(* LS Electric XG5000 project: XMC_SingleAxis_FBs *)
(* sample programs for single axis function blocks. *)
(* PLC LSPLC *)
(* module base 0 slot 0: Input/Output Module:XMC-DN24 (DC 24V Input 8Points/TR output 16Points) *)
(* module base 0 slot 1: Internal Analog Input/Output:XMF-AH04E (A/D voltage/current 2 channels, D/A voltage 2 channels) *)
(* task Periodic Task: Kind=2 *)
(* task Initialization Task: Kind=1 *)
(* task NC Program: Kind=6 *)
VAR_GLOBAL
    ContinuousRelative_INST : MC_MOVECONTINUOUSRELATIVE; (* MC_MoveContinuousRelative fb *)
    Relative_INST : MC_MOVECONTINUOUSRELATIVE; (* MC_MoveContinuousRelative fb *)
END_VAR

PROGRAM ECAT_Connect_Example (* task: Scan Program *)
(* example of LS_Connect and LS_Disconnect function blocks *)
VAR
    Execute_Connect : BOOL; (* Execute LS_Connect function block *)
    Execute_Disconnect : BOOL; (* Execute LS_Disconnect *)
    INST_LS_CONNECT : LS_CONNECT; (* Instance of LS_Connect function block *)
    INST_LS_DISCONNECT : LS_DISCONNECT; (* LS_Disconnect function block instance *)
END_VAR
(* AutomationDirect.com has provided this code for convenience. This sample code is provided "as-is" with no expressed or implied warranty. 
 If the end user includes any of the sample code (in whole or part), it is the user's responsibility to completely modify, integrate, and test any code to ensure it meets all system and 
 safety requirements for the intended application or system. *)

//Example of LS_Connect Function block to connect EtherCAT network
INST_LS_CONNECT(Execute:=Execute_Connect, ErrorID=>INST_LS_CONNECT.ErrorID);

//Example of LS_Disconnect Function block to disconnect the EtherCAT network
INST_LS_DISCONNECT(Execute:=Execute_Disconnect, ErrorID=>INST_LS_DISCONNECT.ErrorID);
END_PROGRAM

PROGRAM MC_Power_Example (* task: Scan Program *)
(* ST example of MC_Power *)
VAR
    Axis1 : UINT; (* axis 1 reference variable *)
    Enable_Power : BOOL; (* command to enable axis power *)
    INST_MC_POWER : MC_POWER; (* MC_Power fb *)
END_VAR
//Set Axis 1 reference
Axis1 := 1;

//Example MC_Power FB.  Check that axis is ready
IF (_AX01_RDY) THEN
	INST_MC_POWER(Enable:=Enable_Power, Axis:=Axis1, ErrorID=>INST_MC_POWER.ErrorID);
END_IF;
END_PROGRAM

PROGRAM Home_Example (* task: Scan Program *)
(* ST example of MC_Home and LS_Home *)
VAR
    Axis1 : UINT; (* axis1 reference variable *)
    Execute_LSHome : BOOL; (* execute LS_Home fb *)
    Execute_MCHome : BOOL; (* execute MC_Home fb *)
    INST_LS_HOME : LS_HOME; (* LS_Home function block *)
    INST_MC_HOME : MC_HOME; (* MC_Home fb *)
END_VAR
//Set Axis1 reference variable
Axis1 := 1;

//check that axis 1 is ready
IF (_AX01_RDY) AND (_AX01_SV_ON) THEN
	
	//Example MC_Home fb
	INST_MC_HOME(Execute:=Execute_MCHome, Axis:=Axis1, Position:=INST_MC_HOME.Position, BufferMode:=0, ErrorID=>INST_MC_HOME.ErrorID);
	
	//Example LS_Home fb
	INST_LS_HOME(Execute:=Execute_LSHome, Axis:=Axis1, Position:=INST_LS_HOME.Position, HomingMethod:=INST_LS_HOME.HomingMethod, 
		SwitchSearchSpeed:=INST_LS_HOME.SwitchSearchSpeed, ZeroSearchSpeed:=INST_LS_HOME.ZeroSearchSpeed, HomingAcc:=INST_LS_HOME.HomingAcc, 
		HomeOffset:=INST_LS_HOME.HomeOffset, DoneBehavior:=INST_LS_HOME.DoneBehavior, BufferMode:=0, ErrorID=>INST_LS_HOME.ErrorID);
END_IF;
END_PROGRAM

PROGRAM MCStop_MCHalt_Example (* task: Scan Program *)
(* ST example for MC_Stop and MC_Halt fb *)
VAR
    Axis1 : UINT; (* reference variable for axis1 *)
    Execute_MCHalt : BOOL; (* Execute MC_Halt fb *)
    Execute_MCStop : BOOL; (* execute MC_Stop fb *)
    INST_MC_HALT : MC_HALT; (* MC_Halt fb *)
    INST_MC_STOP : MC_STOP; (* MC_Stop function block *)
END_VAR
//Set reference for axis
Axis1 := 1;

//check that axes are ready
IF (_AX01_RDY) AND (_AX01_SV_ON) THEN
	//Example of MC_Stop fb
	INST_MC_STOP(Execute:=Execute_MCStop, Axis:=Axis1, Deceleration:=50000.0, Jerk:=1000.0, ErrorID=>INST_MC_STOP.ErrorID);
	
	//Example of MC_Halt fb
	INST_MC_HALT(Execute:=Execute_MCHalt, Axis:=Axis1, Deceleration:=50000.0, Jerk:=1000.0, BufferMode:=0,ErrorID=>INST_MC_HALT.ErrorID);
END_IF;
END_PROGRAM

PROGRAM Read_Status_FBs (* task: Scan Program *)
(* ST example for MC fbs that read axis status *)
VAR
    Axis1 : UINT; (* reference for axis 1 *)
    Enable_ReadActualPosition : BOOL; (* enable MC_ReadActualPosition fb *)
    Enable_ReadActualTorque : BOOL; (* Enable MC_ReadActualTorque fb *)
    Enable_ReadActualVelocity : BOOL; (* enable MC_ReadActualVelocity fb *)
    Enable_ReadCommandedPosition : BOOL; (* enable MC_ReadCommandedPosition *)
    Enable_ReadCommandedTorque : BOOL; (* enable MC_ReadCommandedTorque fb *)
    Enable_ReadCommandedVelocity : BOOL; (* enable MC_ReadCommandedVelocity fb *)
    Enable_ReadMotionInfo : BOOL; (* Enable MC_ReadMotionInfo fb *)
    INST_READACTUALPOSITION : MC_READACTUALPOSITION; (* MC_ReadActualPosition fb *)
    INST_READACTUALTORQUE : MC_READACTUALTORQUE; (* MC_ReadActualTorque function block *)
    INST_READACTUALVELOCITY : MC_READACTUALVELOCITY; (* MC_ReadActualVelocity fb *)
    INST_READCOMMANDEDPOSITION : MC_READCOMMANDEDPOSITION; (* MC_ReadCommandedPosition fb *)
    INST_READCOMMANDEDTORQUE : MC_READCOMMANDEDTORQUE; (* MC_ReadCommandedTorque fb *)
    INST_READCOMMANDEDVELOCITY : MC_READCOMMANDEDVELOCITY; (* MC_ReadCommandedVelocity fb *)
    INST_READMOTIONINFO : MC_READMOTIONINFO; (* MC_ReadMotionInfo fb *)
END_VAR
//Set Axis Reference
Axis1 := 1;

IF (_AX01_RDY) THEN
	//Example of MC_ReadMotionInfo
	INST_READMOTIONINFO(Enable:=Enable_ReadMotionInfo, Axis:=Axis1, ParameterNumber:=INST_READMOTIONINFO.ParameterNumber, ErrorID=>INST_READMOTIONINFO.ErrorID);
	
	//Example of MC_ReadActualPosition
	INST_READACTUALPOSITION(Enable:=Enable_ReadActualPosition, Axis:=Axis1, ErrorID=>INST_READACTUALPOSITION.ErrorID);
	
	//Example of MC_ReadActualVelocity
	INST_READACTUALVELOCITY(Enable:=Enable_ReadActualVelocity, Axis:=Axis1, ErrorID=>INST_READACTUALVELOCITY.ErrorID);
	
	//Example of MC_ReadActualTorque
	INST_READACTUALTORQUE(Enable:=Enable_ReadActualTorque, Axis:=Axis1, ErrorID=>INST_READACTUALTORQUE.ErrorID);
	
	//Example of MC_ReadCommandedPosition
	INST_READCOMMANDEDPOSITION(Enable:=Enable_ReadCommandedPosition, Axis:=Axis1,ErrorID=>INST_READCOMMANDEDPOSITION.ErrorID);
	
	//Example of MC_ReadCommandedVelocity
	INST_READCOMMANDEDVELOCITY(Enable:=Enable_ReadCommandedVelocity, Axis:=Axis1, ErrorID=>INST_READCOMMANDEDVELOCITY.ErrorID);
	
	//Example MC_ReadCommandedTorque
	INST_READCOMMANDEDTORQUE(Enable:=Enable_ReadCommandedTorque, Axis:=Axis1, ErrorID=>INST_READCOMMANDEDTORQUE.ErrorID);
	
END_IF;
END_PROGRAM

PROGRAM MC_Reset_Example (* task: Scan Program *)
(* ST example for MC_Reset & MC_Reset2 *)
VAR
    Axis1 : UINT; (* reference variable for axis1 *)
    Execute_MCReset : BOOL; (* execute MC_Reset fb *)
    Execute_MCReset2 : BOOL; (* Execute MC_Reset2 fb *)
    INST_MC_RESET : MC_RESET; (* MC_Reset fb *)
    INST_MC_RESET2 : MC_RESET2; (* MC_Reset2 fb *)
END_VAR
//Set Axis Reference
Axis1 := 1;

IF (_AX01_RDY) THEN
	//Example of MC_Reset
	INST_MC_RESET(Execute:=Execute_MCReset, Axis:=Axis1, ErrorType:=INST_MC_RESET.ErrorType, ErrorID=>INST_MC_RESET.ErrorID);
	
	INST_MC_RESET2(Execute:=Execute_MCReset2, Axis:=Axis1, ErrorType:=INST_MC_RESET2.ErrorType, ErrorID=>INST_MC_RESET2.ErrorID);
	
END_IF;
END_PROGRAM

PROGRAM MC_MoveAbsolute_Example (* task: Scan Program *)
(* example of MC_MoveAbsolute *)
VAR
    Axis1 : UINT; (* axis 1 reference variable *)
    Execute_MoveAbsolute : BOOL; (* execute MC_MoveAbsolute *)
    INST_MOVEABSOLUTE : MC_MOVEABSOLUTE; (* MC_MoveAbsolute fb *)
END_VAR
//Set axis reference
Axis1 := 1;

IF (_AX01_RDY) AND (_AX01_SV_ON) AND (_AX01_HOME_CMPL) THEN
	//Example of MC_MoveAbsolute
	INST_MOVEABSOLUTE(Execute:=Execute_MoveAbsolute, Axis:=Axis1, ContinuousUpdate:=0, Position:=INST_MOVEABSOLUTE.Position, 
		Velocity:=INST_MOVEABSOLUTE.Velocity, Acceleration:=INST_MOVEABSOLUTE.Acceleration, Deceleration:=INST_MOVEABSOLUTE.Deceleration, 
		Jerk:=INST_MOVEABSOLUTE.Jerk, Direction:=INST_MOVEABSOLUTE.Direction, BufferMode:=0, ErrorID=>INST_MOVEABSOLUTE.ErrorID);
END_IF;
END_PROGRAM

PROGRAM MC_MoveRelative_Example (* task: Scan Program *)
(* ST example for MC_MoveRelative fb *)
VAR
    Axis1 : UINT; (* reference for Axis1 *)
    Execute_MoveRelative : BOOL; (* execute MC_MoveRelative fb *)
    INST_MOVERELATIVE : MC_MOVERELATIVE; (* MC_MoveRelative fb *)
END_VAR
//Set axis reference
Axis1 := 1;

IF (_AX01_RDY) AND (_AX01_SV_ON) THEN
	//Example of MC_MoveRelative
	INST_MOVERELATIVE(Execute:=Execute_MoveRelative, Axis:=Axis1, ContinuousUpdate:=0, Distance:=INST_MOVERELATIVE.Distance,
		 Velocity:=INST_MOVERELATIVE.Velocity, Acceleration:=INST_MOVERELATIVE.Acceleration, Deceleration:=INST_MOVERELATIVE.Deceleration, 
		 Jerk:=INST_MOVERELATIVE.Jerk, BufferMode:=0, ErrorID=>INST_MOVERELATIVE.ErrorID);	
END_IF;
END_PROGRAM

PROGRAM MC_MoveAdditive_Example (* task: Scan Program *)
(* ST example for MC_MoveAdditive fb *)
VAR
    Axis1 : UINT; (* axis 1 reference variable *)
    Execute_MoveAdditive : BOOL; (* execute MC_MoveAdditive fb *)
    INST_MOVEADDITIVE : MC_MOVEADDITIVE; (* MC_MoveAdditive fb *)
END_VAR
//Set axis reference
Axis1 := 1;

IF (_AX01_RDY) AND (_AX01_SV_ON) AND (_AX01_HOME_CMPL) THEN
	//Example of MC_MoveAdditive
	INST_MOVEADDITIVE(Execute:=Execute_MoveAdditive, Axis:=Axis1, ContinuousUpdate:=0, Distance:=INST_MOVEADDITIVE.Distance, 
		Velocity:=INST_MOVEADDITIVE.Velocity, Acceleration:=INST_MOVEADDITIVE.Acceleration, Deceleration:=INST_MOVEADDITIVE.Deceleration, 
		Jerk:=INST_MOVEADDITIVE.Jerk, BufferMode:=0, ErrorID=>INST_MOVEADDITIVE.ErrorID);
END_IF;
END_PROGRAM

PROGRAM MC_MoveVelocity_Example (* task: Scan Program *)
(* ST example for MC_MoveVelocity fb *)
VAR
    Axis1 : UINT; (* axis 1 reference variable *)
    Execute_MoveVelocity : BOOL; (* execute MC_MoveVelocity fb *)
    INST_MOVEVELOCITY : MC_MOVEVELOCITY; (* MC_MoveVelocity fb *)
END_VAR
//Set axis reference
Axis1 := 1;

IF (_AX01_RDY) AND (_AX01_SV_ON)  THEN
	//Example MC_MoveVelocity fb
	INST_MOVEVELOCITY(Execute:=Execute_MoveVelocity, Axis:=Axis1, ContinuousUpdate:=0, Velocity:=INST_MOVEVELOCITY.Velocity, 
		Acceleration:=INST_MOVEVELOCITY.Acceleration, Deceleration:=INST_MOVEVELOCITY.Deceleration, Jerk:=INST_MOVEVELOCITY.Jerk, 
		Direction:=INST_MOVEVELOCITY.Direction, BufferMode:=0, ErrorID=>INST_MOVEVELOCITY.ErrorID);
END_IF;
END_PROGRAM

PROGRAM MC_MoveContinuousAbsolute_Example (* task: Scan Program *)
(* ST example of MC_MoveContinuousAbsolute fb *)
VAR
    Axis1 : UINT; (* axis 1 reference variable *)
    Execute_MoveContAbs : BOOL; (* execute MC_MoveContinuousAbsolute fb *)
    INST_MOVECONTINUOUSABSOLUTE : MC_MOVECONTINUOUSABSOLUTE; (* MC_MoveContinuousAbsolute fb *)
END_VAR
//Set axis reference
Axis1 := 1;

IF (_AX01_RDY) AND (_AX01_SV_ON)  AND (_AX01_HOME_CMPL) THEN
	//Example MC_MoveContinuousAbsolute fb
	INST_MOVECONTINUOUSABSOLUTE(Execute:=Execute_MoveContAbs, Axis:=Axis1, ContinuousUpdate:=0, Position:=INST_MOVECONTINUOUSABSOLUTE.Position, 
		EndVelocity:=INST_MOVECONTINUOUSABSOLUTE.EndVelocity, Velocity:=INST_MOVECONTINUOUSABSOLUTE.Velocity, Acceleration:=INST_MOVECONTINUOUSABSOLUTE.Acceleration, 
		Deceleration:=INST_MOVECONTINUOUSABSOLUTE.Deceleration, Jerk:=INST_MOVECONTINUOUSABSOLUTE.Jerk, Direction:=INST_MOVECONTINUOUSABSOLUTE.Direction, 
		BufferMode:=0, ErrorID=>INST_MOVECONTINUOUSABSOLUTE.ErrorID);
END_IF;
END_PROGRAM

PROGRAM MC_MoveContinuousRelative_Example (* task: Scan Program *)
(* ST example for MC_MoveContinuousRelative fb *)
VAR
    Axis1 : UINT; (* axis 1 reference variable *)
    Execute_MoveContRel : BOOL; (* execute MC_MoveContinuousRelative fb *)
    INST_MOVECONTINUOUSRELATIVE : MC_MOVECONTINUOUSRELATIVE; (* MC_MoveContinuousRelative fb *)
END_VAR
//Set axis reference
Axis1 := 1;

IF (_AX01_RDY) AND (_AX01_SV_ON) THEN
	//Example MC_MoveContinuousRelative fb
	INST_MOVECONTINUOUSRELATIVE(Execute:=Execute_MoveContRel, Axis:=Axis1, ContinuousUpdate:=0, Distance:=INST_MOVECONTINUOUSRELATIVE.Distance, 
		EndVelocity:=INST_MOVECONTINUOUSRELATIVE.EndVelocity, Velocity:=INST_MOVECONTINUOUSRELATIVE.Velocity, Acceleration:=INST_MOVECONTINUOUSRELATIVE.Acceleration, 
		Deceleration:=INST_MOVECONTINUOUSRELATIVE.Deceleration, Jerk:=INST_MOVECONTINUOUSRELATIVE.Jerk, 
		BufferMode:=0, ErrorID=>INST_MOVECONTINUOUSRELATIVE.ErrorID);
END_IF;
END_PROGRAM

PROGRAM MC_TorqueControl_Example (* task: Scan Program *)
(* ST example for MC_TorqueControl fb *)
VAR
    Axis1 : UINT; (* axis 1 reference variable *)
    Execute_TrqControl : BOOL; (* Execute MC_TorqueControl fb *)
    INST_TORQUECONTROL : MC_TORQUECONTROL; (* MC_TorqueControl fb *)
END_VAR
//Set axis reference
Axis1 := 1;

IF (_AX01_RDY) AND (_AX01_SV_ON) THEN
	//Example MC_TorqueControl fb
	INST_TORQUECONTROL(Execute:=Execute_TrqControl, Axis:=Axis1, ContinuousUpdate:=0, Torque:=INST_TORQUECONTROL.Torque, 
		TorqueRamp:=INST_TORQUECONTROL.TorqueRamp, Velocity:=INST_TORQUECONTROL.Velocity, Acceleration:=INST_TORQUECONTROL.Acceleration, 
		Deceleration:=INST_TORQUECONTROL.Deceleration, Jerk:=INST_TORQUECONTROL.Jerk, Direction:=INST_TORQUECONTROL.Direction, 
		BufferMode:=0, ErrorID=>INST_TORQUECONTROL.ErrorID);
END_IF;
END_PROGRAM

PROGRAM MC_SetPosition_Example (* task: Scan Program *)
(* ST example of MC_SetPosition *)
VAR
    Axis1 : UINT; (* axis 1 reference variable *)
    Execute_SetPosition : BOOL; (* execute MC_SetPosition fb *)
    INST_SETPOSITION : MC_SETPOSITION; (* MC_SetPositionFB *)
END_VAR
//Set axis reference
Axis1 := 1;

IF (_AX01_RDY) AND (_AX01_SV_ON) THEN
	//Example MC_SetPosition fb
	INST_SETPOSITION(Execute:=Execute_SetPosition, Axis:=Axis1, Position:=INST_SETPOSITION.Position, Relative:=INST_SETPOSITION.Relative, 
		ExecutionMode:=INST_SETPOSITION.ExecutionMode, ErrorID=>INST_SETPOSITION.ErrorID);
END_IF;
END_PROGRAM

PROGRAM MC_SetOverride_Example (* task: Scan Program *)
(* ST example of MC_SetOverride fb *)
VAR
    Axis1 : UINT; (* axis 1 reference variable *)
    Execute_Override : BOOL; (* execute MC_SetOverride *)
    INST_SETOVERRIDE : MC_SETOVERRIDE; (* MC_SetOverride fb *)
END_VAR
//Set axis reference
Axis1 := 1;

IF (_AX01_RDY) AND (_AX01_SV_ON) THEN
	//Example MC_SetOverride fb
	INST_SETOVERRIDE(Enable:=Execute_Override, Axis:=Axis1, VelFactor:=INST_SETOVERRIDE.VelFactor, AccFactor:=INST_SETOVERRIDE.AccFactor, 
		JerkFactor:=INST_SETOVERRIDE.JerkFactor, ErrorID=>INST_SETOVERRIDE.ErrorID);
END_IF;
END_PROGRAM

PROGRAM Read_Write_Parameters (* task: Scan Program *)
(* ST example for MC_ReadParameter and MC_WriteParameter *)
VAR
    Axis1 : UINT; (* axis 1 reference variable *)
    Execute_Read : BOOL; (* Execute MC_ReadParameter fb *)
    Execute_Write : BOOL; (* execute MC_WriteParameter *)
    INST_READPARAMETER : MC_READPARAMETER; (* MC_ReadParameter fb *)
    INST_WRITEPARAMETER : MC_WRITEPARAMETER; (* MC_WriteParameter fb *)
END_VAR
//Set axis reference
Axis1 := 1;

IF (_AX01_RDY) THEN
	//Example of MC_ReadParameter fb
	INST_READPARAMETER(Enable:=Execute_Read, Axis:=Axis1, ParameterNumber:=INST_READPARAMETER.ParameterNumber, 
		ErrorID=>INST_READPARAMETER.ErrorID, Value=>INST_READPARAMETER.Value);
		
	
	//Example of MC_WriteParameter fb
	INST_WRITEPARAMETER(Execute:=Execute_Write, Axis:=Axis1, ParameterNumber:=INST_WRITEPARAMETER.ParameterNumber, Value:=INST_WRITEPARAMETER.Value, 
		ExecutionMode:=INST_WRITEPARAMETER.ExecutionMode, ErrorID=>INST_WRITEPARAMETER.ErrorID);	
		
END_IF;
END_PROGRAM

PROGRAM MC_TouchProbe_Example (* task: Scan Program *)
(* ST example of MC_TouchProbe and MC_TouchProbeEx *)
VAR
    Axis1 : UINT; (* axis 1 reference *)
    Execute_TouchProbe : BOOL; (* execute MC_TouchProbe *)
    Execute_TouchProveEx : BOOL; (* execute MC_TouchProbeEX fb *)
    INST_TOUCHPROBE : MC_TOUCHPROBE; (* MC_TouchProbe fb *)
    INST_TOUCHPROBEEX : MC_TOUCHPROBEEX; (* MC_TouchProbeEx fb *)
END_VAR
//Set axis reference
Axis1 := 1;

IF (_AX01_RDY) AND (_AX01_SV_ON) THEN
	//Example MC_TouchProbel fb
	INST_TOUCHPROBE(Execute:=Execute_TouchProbe, Axis:=Axis1, TriggerInput:=INST_TOUCHPROBE.TriggerInput, WindowOnly:=INST_TOUCHPROBE.WindowOnly, 
		FirstPosition:=INST_TOUCHPROBE.FirstPosition, LastPosition:=INST_TOUCHPROBE.LastPosition, 
		ErrorID=>INST_TOUCHPROBE.ErrorID, RecordedPosition=>INST_TOUCHPROBE.RecordedPosition);
		
	
	//Exampe of MC_TouchProbeEX fb
	INST_TOUCHPROBEEX(Execute:=Execute_TouchProveEx, Axis:=Axis1, TriggerInput:=INST_TOUCHPROBEEX.TriggerInput, TriggerMode:=INST_TOUCHPROBEEX.TriggerMode, 
		WindowOnly:=INST_TOUCHPROBEEX.WindowOnly, FirstPosition:=INST_TOUCHPROBEEX.FirstPosition, LastPosition:=INST_TOUCHPROBEEX.LastPosition, 
		ErrorID=>INST_TOUCHPROBEEX.ErrorID, RecordedPosition=>INST_TOUCHPROBEEX.RecordedPosition);
		
END_IF;
END_PROGRAM

PROGRAM MC_AbortTrigger_Example (* task: Scan Program *)
(* ST example MC_AbortTrigger fb *)
VAR
    Axis1 : UINT; (* axis 1 reference *)
    Execute_AbortTrigger : BOOL; (* execute MC_AbortTrigger fb *)
    INST_ABORTTRIGGER : MC_ABORTTRIGGER; (* MC_AbortTrigger fb *)
END_VAR
//Set axis reference
Axis1 := 1;

IF (_AX01_RDY) AND (_AX01_SV_ON) THEN
	//Example MC_AbortTrigger fb
	INST_ABORTTRIGGER(Execute:=Execute_AbortTrigger, Axis:=Axis1, TriggerInput:=INST_ABORTTRIGGER.TriggerInput, ErrorID=>INST_ABORTTRIGGER.ErrorID);
END_IF;
END_PROGRAM

PROGRAM MC_SuperImposed_Example (* task: Scan Program *)
(* ST example of MC_SuperImposed and MC_HaltSuperImposed *)
VAR
    Axis1 : UINT; (* axis 1 reference *)
    Execute_HaltSuperImposed : BOOL; (* execute MC_HaltSuperImposed fb *)
    Execute_SuperImposed : BOOL; (* execute MC_MoveSuperImposed *)
    INST_HALTSUPERIMPOSED : MC_HALTSUPERIMPOSED; (* MC_HaltSuperImposed *)
    INST_MOVESUPERIMPOSED : MC_MOVESUPERIMPOSED; (* MC_MoveSuperImposed fb *)
END_VAR
//Set axis reference
Axis1 := 1;

IF (_AX01_RDY) AND (_AX01_SV_ON) THEN
	//Example MC_MoveSuperImposed fb
	INST_MOVESUPERIMPOSED(Execute:=Execute_SuperImposed, Axis:=Axis1, ContinuousUpdate:=0, Distance:=INST_MOVESUPERIMPOSED.Distance, 
		VelocityDiff:=INST_MOVESUPERIMPOSED.VelocityDiff, Acceleration:=INST_MOVESUPERIMPOSED.Acceleration, 
		Deceleration:=INST_MOVESUPERIMPOSED.Deceleration, Jerk:=INST_MOVESUPERIMPOSED.Jerk, ErrorID=>INST_MOVESUPERIMPOSED.ErrorID, 
		CoveredDistance=>INST_MOVESUPERIMPOSED.CoveredDistance);
		
	//MC_HaltSuperImposed
	INST_HALTSUPERIMPOSED(Execute:=Execute_HaltSuperImposed, Axis:=Axis1, Deceleration:=INST_HALTSUPERIMPOSED.Deceleration, 
		Jerk:=INST_HALTSUPERIMPOSED.Jerk, ErrorID=>INST_HALTSUPERIMPOSED.ErrorID)	;
		
END_IF;
END_PROGRAM